// TIA Portal project "Palitizer" (V16)
// Vorlageprojekt für das Buch mit Zielsystem S7-1200

(* hardware
DEVICE "S7-1200-Station_1"  S7-1200 Station
   slot 0: "Baugruppenträger_0"  Rack  V1.0
   slot 1: "PLC_1"  CPU 1211C DC/DC/DC  6ES7 211-1AE40-0XB0  V4.1
DEVICE "HMI_1"  KTP700 Basic PN
   slot 0: "HMI_1"  KTP700 Basic PN  6AV2 123-2GB03-0AX0  16.0.0.0
   slot 1: "HMI_RT_1"  KTP700 Basic PN  6AV2 123-2GB03-0AX0  16.0.0.0
   slot 5: "HMI_1.IE_CP_1"  PROFINET Interface  16.0.0.0
      slot 1: "PROFINET Interface_1"  PROFINET Interface
         slot 1: "Port_1"  Port
*)

// ===== PLC "PLC_1"  CPU 1211C DC/DC/DC =====

VAR_GLOBAL   // PLC tag table "Standard-Variablentabelle"
   "I_Auto" AT %I0.0 : Bool;
   "I_Manual" AT %I0.1 : Bool;
   "I_Start" AT %I0.2 : Bool;
   "I_Stop" AT %I0.3 : Bool;
   "I_E_Stop" AT %I0.4 : Bool;
   "Q_Start_Light" AT %Q0.0 : Bool;
   "Q_Stop_Light" AT %Q0.1 : Bool;
   "M_Machine_Running" AT %M0.0 : Bool;
   "I_Pallet_Loaded" AT %I1.3 : Bool;   // Sensor ON the elevator. Goes TRUE when pallet is in position.
   "Q_Pallet_Feeder" AT %Q1.5 : Bool;   // The conveyor belt bringing pallets to the machine.
   "Q_Load_Pallet" AT %Q1.6 : Bool;   // The motorized rollers ON the elevator itself.
   "Q_Pallets_Emitter" AT %Q2.1 : Bool;   // Q_Pallets_Emitter
   "I_Box_At_Entry" AT %I0.6 : Bool;   // Photo-eye sensor that detects boxes passing.
   "I_Clamped" AT %I0.7 : Bool;   // Sensor confirming the clamp is fully closed.
   "Q_Box_Feeder" AT %Q0.4 : Bool;   // First conveyor bringing boxes in.
   "Q_Load_Belt" AT %Q0.5 : Bool;   // Second conveyor pushing boxes into the clamping area.
   "Q_Clamp" AT %Q0.7 : Bool;   // Pneumatic clamp to hold the row of boxes.
   "Q_Parts_Emitter" AT %Q2.0 : Bool;   // Spawns boxes in Factory I/O.
   "M_Box_Edge_Mem" AT %M0.1 : Bool;
   "M_Row_Ready" AT %M0.2 : Bool;
   "M_Reset_Row" AT %M0.3 : Bool;
   "Q_Push" AT %Q1.1 : Bool;   // Pushes clamped row onto plate
   "I_pusher_limit" AT %I1.0 : Bool;
   "Q_Open_Plate" AT %Q1.2 : Bool;
   "I_Plate_Limit" AT %I1.4 : Bool;
   "Q_Elevator_Up" AT %Q1.3 : Bool;
   "Q_Move_to_Limit" AT %Q1.4 : Bool;
   "I_Reset" AT %I1.5 : Bool;
   "Q_Elevator_down" AT %Q1.0 : Bool;
   "M_Eject_Pallet" AT %M0.4 : Bool;
   "I_Elevator_Moving" AT %I0.5 : Bool;
   "Q_Turn" AT %Q0.6 : Bool;
   "Q_Remover" AT %Q2.2 : Bool;
   "Q_Exit_Conveyor" AT %Q1.7 : Bool;
   "M_Target_Boxes" AT %MW10 : Int;   // Tells the counter how many boxes to wait for.
   "M_Target_Rows" AT %MW12 : Int;   // Tells the sequencer how many rows to push.
   "M_Enable_Turn" AT %M1.0 : Bool;   // Flag to activate the Turn actuator.
   "M_Machine_Fault" AT %M1.1 : Bool;
   "M_Cmd_Run" AT %M1.2 : Bool;
   "System_Byte" AT %MB5 : Byte;
   "FirstScan" AT %M5.0 : Bool;
   "DiagStatusUpdate" AT %M5.1 : Bool;
   "AlwaysTRUE" AT %M5.2 : Bool;
   "AlwaysFALSE" AT %M5.3 : Bool;
   "Clock_Byte" AT %MB2 : Byte;
   "Clock_10Hz" AT %M2.0 : Bool;
   "Clock_5Hz" AT %M2.1 : Bool;
   "Clock_2.5Hz" AT %M2.2 : Bool;
   "Clock_2Hz" AT %M2.3 : Bool;
   "Clock_1.25Hz" AT %M2.4 : Bool;
   "Clock_1Hz" AT %M2.5 : Bool;
   "Clock_0.625Hz" AT %M2.6 : Bool;
   "Clock_0.5Hz" AT %M2.7 : Bool;
   "Q_faulted" AT %Q0.2 : Bool;
   "Q_Warning_light" AT %Q2.3 : Bool;
   "negative_box_at_entry" AT %M0.5 : Bool;
   "Cmd_Push_Auto" AT %M0.6 : Bool;
   "Cmd_Push_Manual" AT %M0.7 : Bool;
   "Cmd_Clamp_Auto" AT %M3.0 : Bool;
   "Cmd_Clamp_Manual" AT %M3.1 : Bool;
   "Cmd_Plate_Auto" AT %M3.2 : Bool;
   "Cmd_Plate_Manual" AT %M3.3 : Bool;
   "Cmd_BoxFeed_Auto" AT %M3.4 : Bool;
   "Cmd_PalletFeed_Auto" AT %M3.5 : Bool;
   "Cmd_ExitConv_Auto" AT %M3.6 : Bool;
   "Cmd_BoxFeed_Manual" AT %M3.7 : Bool;
   "Cmd_PalletFeed_Manual" AT %M4.0 : Bool;
   "Cmd_ExitConv_Manual" AT %M4.1 : Bool;
   "Cmd_ElevUp_Auto" AT %M4.2 : Bool;
   "Cmd_ElevUp_Manual" AT %M4.3 : Bool;
   "Cmd_ElevDown_Auto" AT %M4.4 : Bool;
   "Cmd_ElevDown_Manual" AT %M4.5 : Bool;
   "System_Byte(1)" AT %MB1 : Byte;
   "Cmd_Turn_Auto" AT %M4.6 : Bool;
   "Cmd_Turn_Manual" AT %M4.7 : Bool;
   "I_Pallet_at_Entry" AT %I1.1 : Bool;
END_VAR

TYPE "UDT_SysCommand"
   STRUCT
      xSwAuto : Bool;
      xSwManual : Bool;
      xBtnStart : Bool;
      xBtnStop : Bool;
      xBtnReset : Bool;
      xEStop_OK : Bool;
      xHmiResetCounters : Bool;
      xHmiAckFault : Bool;
   END_STRUCT;
END_TYPE

TYPE "UDT_SysStatus"
   STRUCT
      xModeAuto : Bool;
      xModeManual : Bool;
      xRunning : Bool;
      xPaused : Bool;
      xFaulted : Bool;
      iStateID : Int;
      iCurrentLayer : Int;
      iTargetLayers : Int;
      iTotalBoxes : DInt;
      iTotalPallets : DInt;
      wAlarmWord : Word;
   END_STRUCT;
END_TYPE

DATA_BLOCK "FB1_Pallet_Handling_DB"   // DB1
{ S7_Optimized_Access := 'TRUE' }
VERSION : 0.1
// stored: InstanceOfName FB1_Pallet_Handling
"FB1_Pallet_Handling"
BEGIN
END_DATA_BLOCK

DATA_BLOCK "FB2_Box_Grouping_DB"   // DB3
{ S7_Optimized_Access := 'TRUE' }
VERSION : 0.1
// stored: InstanceOfName FB2_Box_Grouping
"FB2_Box_Grouping"
BEGIN
END_DATA_BLOCK

DATA_BLOCK "FB3_Elevator_Stacker_DB"   // DB5
{ S7_Optimized_Access := 'TRUE' }
VERSION : 0.1
// stored: InstanceOfName FB3_Elevator_Stacker
"FB3_Elevator_Stacker"
BEGIN
END_DATA_BLOCK

DATA_BLOCK "FB_ModeManager_DB"   // DB11
{ S7_Optimized_Access := 'TRUE' }
VERSION : 0.1
// stored: InstanceOfName FB_ModeManager
"FB_ModeManager"
BEGIN
END_DATA_BLOCK

DATA_BLOCK "DB_Machine"   // DB12
{ S7_Optimized_Access := 'FALSE' }
VERSION : 0.1
   VAR
      Cmd : "UDT_SysCommand";
      Sts : "UDT_SysStatus";
   END_VAR
BEGIN
END_DATA_BLOCK

DATA_BLOCK "InstDB_Cylinder_Pusher"   // DB13
{ S7_Optimized_Access := 'TRUE' }
VERSION : 0.1
// stored: InstanceOfName FB_Cylinder
"FB_Cylinder"
BEGIN
   i_xInterlock := true;
END_DATA_BLOCK

DATA_BLOCK "InstDB_Cyl_Clamp"   // DB14
{ S7_Optimized_Access := 'TRUE' }
VERSION : 0.1
// stored: InstanceOfName FB_Cylinder
"FB_Cylinder"
BEGIN
END_DATA_BLOCK

DATA_BLOCK "InstDB_Cyl_Plate"   // DB15
{ S7_Optimized_Access := 'TRUE' }
VERSION : 0.1
// stored: InstanceOfName FB_Cylinder
"FB_Cylinder"
BEGIN
END_DATA_BLOCK

DATA_BLOCK "FB_Motor_BoxFeed"   // DB16
{ S7_Optimized_Access := 'TRUE' }
VERSION : 0.1
// stored: InstanceOfName FB_Motor
"FB_Motor"
BEGIN
   i_xThermalFault := true;
END_DATA_BLOCK

DATA_BLOCK "FB_Motor_PalletFeed"   // DB17
{ S7_Optimized_Access := 'TRUE' }
VERSION : 0.1
// stored: InstanceOfName FB_Motor
"FB_Motor"
BEGIN
   i_xThermalFault := True;
END_DATA_BLOCK

DATA_BLOCK "FB_Motor_ExitConv"   // DB18
{ S7_Optimized_Access := 'TRUE' }
VERSION : 0.1
// stored: InstanceOfName FB_Motor
"FB_Motor"
BEGIN
   i_xThermalFault := true;
END_DATA_BLOCK

DATA_BLOCK "InstDB_Motor_ElevUp"   // DB19
{ S7_Optimized_Access := 'TRUE' }
VERSION : 0.1
// stored: InstanceOfName FB_Motor
"FB_Motor"
BEGIN
   i_xInterlock := true;
   i_xThermalFault := true;
END_DATA_BLOCK

DATA_BLOCK "InstDB_Motor_ElevDown"   // DB20
{ S7_Optimized_Access := 'TRUE' }
VERSION : 0.1
// stored: InstanceOfName FB_Motor
"FB_Motor"
BEGIN
   i_xThermalFault := true;
   i_xInterlock := true;
END_DATA_BLOCK

DATA_BLOCK "InstDB_Cyl_Turn"   // DB21
{ S7_Optimized_Access := 'TRUE' }
VERSION : 0.1
// stored: InstanceOfName FB_Cylinder
"FB_Cylinder"
BEGIN
END_DATA_BLOCK

// folder: System blocks/Program resources

DATA_BLOCK "counter1"   // DB2
{ S7_Optimized_Access := 'TRUE' }
AUTHOR : Simatic
FAMILY : IEC
NAME : CNTR
VERSION : 1.0
// stored: InstanceOfName IEC_COUNTER
"IEC_COUNTER"
BEGIN
END_DATA_BLOCK

DATA_BLOCK "IEC_Timer_0_DB"   // DB4
{ S7_Optimized_Access := 'TRUE' }
AUTHOR : Simatic
FAMILY : IEC
NAME : IEC_TMR
VERSION : 1.0
// stored: InstanceOfName IEC_TIMER
"IEC_TIMER"
BEGIN
END_DATA_BLOCK

DATA_BLOCK "IEC_Timer_0_DB_1"   // DB6
{ S7_Optimized_Access := 'TRUE' }
AUTHOR : Simatic
FAMILY : IEC
NAME : IEC_TMR
VERSION : 1.0
// stored: InstanceOfName IEC_TIMER
"IEC_TIMER"
BEGIN
END_DATA_BLOCK

DATA_BLOCK "IEC_Timer_0_DB_2"   // DB7
{ S7_Optimized_Access := 'TRUE' }
AUTHOR : Simatic
FAMILY : IEC
NAME : IEC_TMR
VERSION : 1.0
// stored: InstanceOfName IEC_TIMER
"IEC_TIMER"
BEGIN
END_DATA_BLOCK

DATA_BLOCK "plate_open"   // DB8
{ S7_Optimized_Access := 'TRUE' }
AUTHOR : Simatic
FAMILY : IEC
NAME : IEC_TMR
VERSION : 1.0
// stored: InstanceOfName IEC_TIMER
"IEC_TIMER"
BEGIN
END_DATA_BLOCK

DATA_BLOCK "plate_close"   // DB9
{ S7_Optimized_Access := 'TRUE' }
AUTHOR : Simatic
FAMILY : IEC
NAME : IEC_TMR
VERSION : 1.0
// stored: InstanceOfName IEC_TIMER
"IEC_TIMER"
BEGIN
END_DATA_BLOCK

DATA_BLOCK "Elevator_Timer"   // DB10
{ S7_Optimized_Access := 'TRUE' }
AUTHOR : Simatic
FAMILY : IEC
NAME : IEC_TMR
VERSION : 1.0
// stored: InstanceOfName IEC_TIMER
"IEC_TIMER"
BEGIN
END_DATA_BLOCK

// folder: (top level)

FUNCTION_BLOCK "FB1_Pallet_Handling"   // FB1, LAD
{ S7_Optimized_Access := 'TRUE' }
VERSION : 0.1
   VAR_INPUT
      i_stState : "UDT_SysStatus";
   END_VAR
BEGIN

REGION Network 1: Spawn Pallets
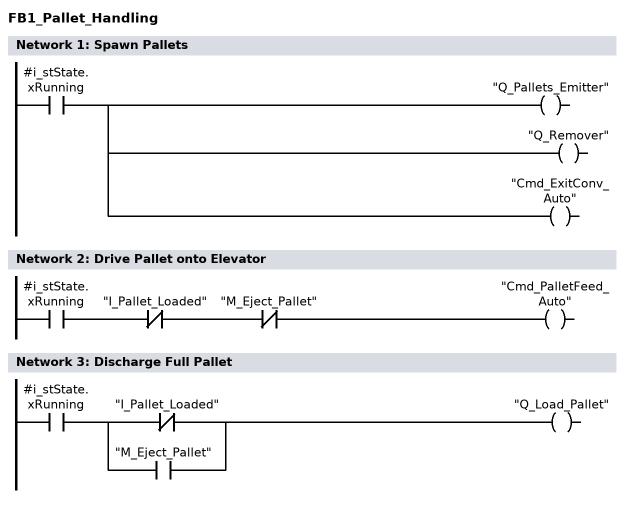
   RUNG wire#powerrail
      Contact( #i_stState.xRunning )
      wire#w1
      Coil( "Q_Pallets_Emitter" )
   END_RUNG
   RUNG wire#w1
      Coil( "Q_Remover" )
   END_RUNG
   RUNG wire#w1
      Coil( "Cmd_ExitConv_Auto" )
   END_RUNG
   // the same network as SCL:
   "Q_Pallets_Emitter" := #i_stState.xRunning;
   "Q_Remover" := #i_stState.xRunning;
   "Cmd_ExitConv_Auto" := #i_stState.xRunning;
END_REGION

REGION Network 2: Drive Pallet onto Elevator
   RUNG wire#powerrail
      Contact( #i_stState.xRunning )
      I_Contact( "I_Pallet_Loaded" )
      I_Contact( "M_Eject_Pallet" )
      Coil( "Cmd_PalletFeed_Auto" )
   END_RUNG
   // the same network as SCL:
   "Cmd_PalletFeed_Auto" := #i_stState.xRunning AND NOT "I_Pallet_Loaded" AND NOT "M_Eject_Pallet";
END_REGION

REGION Network 3: Discharge Full Pallet
   RUNG wire#powerrail
      Contact( #i_stState.xRunning )
      wire#w1
      I_Contact( "I_Pallet_Loaded" )
      wire#w2
      Coil( "Q_Load_Pallet" )
   END_RUNG
   RUNG wire#w1
      Contact( "M_Eject_Pallet" )
   END_RUNG wire#w2
   // the same network as SCL:
   "Q_Load_Pallet" := #i_stState.xRunning AND (NOT "I_Pallet_Loaded" OR "M_Eject_Pallet");
END_REGION
END_FUNCTION_BLOCK

FUNCTION_BLOCK "FB2_Box_Grouping"   // FB2, LAD
{ S7_Optimized_Access := 'TRUE' }
VERSION : 0.1
   VAR_INPUT
      i_stState : "UDT_SysStatus";
      i_stCmd : "UDT_SysCommand";
   END_VAR
   VAR_TEMP   // added for the SCL form of the ladder/FBD networks
      _w1 : Bool;
   END_VAR
BEGIN

REGION Network 1: Spawns boxes in Factory I/O.
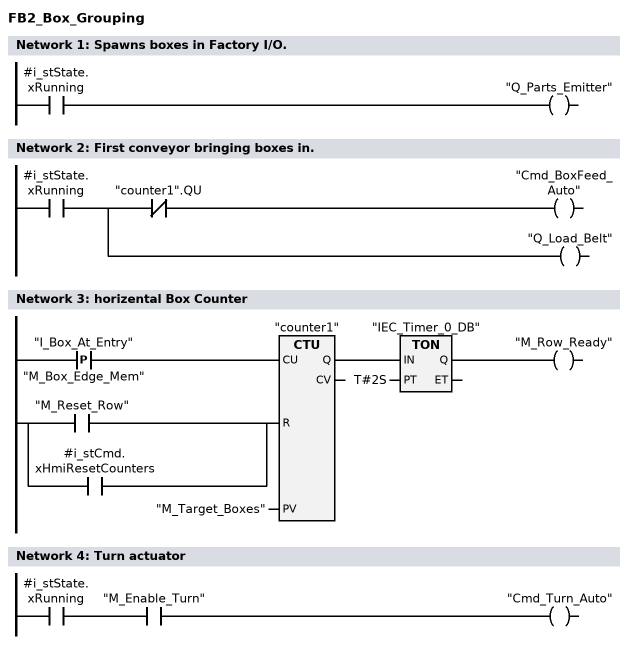
   RUNG wire#powerrail
      Contact( #i_stState.xRunning )
      Coil( "Q_Parts_Emitter" )
   END_RUNG
   // the same network as SCL:
   "Q_Parts_Emitter" := #i_stState.xRunning;
END_REGION

REGION Network 2: First conveyor bringing boxes in.
   RUNG wire#powerrail
      Contact( #i_stState.xRunning )
      wire#w1
      I_Contact( "counter1".QU )
      Coil( "Cmd_BoxFeed_Auto" )
   END_RUNG
   RUNG wire#w1
      Coil( "Q_Load_Belt" )
   END_RUNG
   // the same network as SCL:
   "Cmd_BoxFeed_Auto" := #i_stState.xRunning AND NOT "counter1".QU;
   "Q_Load_Belt" := #i_stState.xRunning;
END_REGION

REGION Network 3: horizental Box Counter
   #_w1 := "I_Box_At_Entry" AND NOT "M_Box_Edge_Mem";   // rising edge of "I_Box_At_Entry"
   "M_Box_Edge_Mem" := "I_Box_At_Entry";
   "counter1".CTU(CU := #_w1, R := "M_Reset_Row" OR #i_stCmd.xHmiResetCounters, PV := "M_Target_Boxes");
   "IEC_Timer_0_DB".TON(IN := "counter1".Q, PT := T#2S);
   "M_Row_Ready" := "IEC_Timer_0_DB".Q;
END_REGION

REGION Network 4: Turn actuator
   RUNG wire#powerrail
      Contact( #i_stState.xRunning )
      Contact( "M_Enable_Turn" )
      Coil( "Cmd_Turn_Auto" )
   END_RUNG
   // the same network as SCL:
   "Cmd_Turn_Auto" := #i_stState.xRunning AND "M_Enable_Turn";
END_REGION
END_FUNCTION_BLOCK

FUNCTION_BLOCK "FB3_Elevator_Stacker"   // FB3, SCL
{ S7_Optimized_Access := 'TRUE' }
VERSION : 0.1
   VAR_INPUT
      i_stState : "UDT_SysStatus";
      i_stCmd : "UDT_SysCommand";
   END_VAR
   VAR_IN_OUT
      io_stState : "UDT_SysStatus";
   END_VAR
   VAR
      stat_Step : Int;
      stat_Retract_Timer : IEC_TIMER;
      stat_Row_Count : Int;
      stat_horizental_box_count : Int;
      stat_vertical_box_count : Int;
      stat_Box_Count : Int;
      stat_Layer_Count : Int;
      stat_Target_Boxes : Int;
      stat_Target_Rows : Int;
      stat_Box_Sensor_Prev : Bool;
      stat_Fault_ID : Int;
      stat_Push_Timeout : IEC_TIMER;
      stat_Plate_Timeout : IEC_TIMER;
      stat_Eject_Timeout : IEC_TIMER;
      push : TON_TIME;
      EjectTimeout : TON_TIME;
   END_VAR
BEGIN
   // --- 1. Fault Reset Logic ---
   // Operator must clear the jam and press Reset to clear the Fault ID
   IF ("I_Reset" OR #i_stCmd.xHmiAckFault)  AND "I_E_Stop" THEN
       #stat_Fault_ID := 0;
       "M_Machine_Fault" := FALSE;
   END_IF;
   // --- 2. Diagnostics & Watchdog Timers ---
   // E-Stop Monitor
   IF NOT "I_E_Stop" THEN
       #stat_Fault_ID := 1;
       #io_stState.xFaulted := TRUE;
       #stat_Step := 0;
   END_IF;
   // Watchdog Timers (Running parallel to the state machine)
   #push(IN:=#stat_Step = 10,
         PT:=T#2.0S);

   #EjectTimeout(IN := #stat_Step = 81,
                 PT := T#8.0S);


   #stat_Plate_Timeout.IN := #stat_Step = 60;
   #stat_Plate_Timeout.PT := T#4.0S;

   // Fault Triggers (If a timer finishes, assign the specific Fault ID)
   IF #push.Q THEN
       #stat_Fault_ID := 2;
       #io_stState.xFaulted := TRUE;
       #stat_Step := 0;
   END_IF;
   IF #stat_Plate_Timeout.Q THEN
       #stat_Fault_ID := 3;
       #io_stState.xFaulted := TRUE;
       #stat_Step := 0;
   END_IF;
   IF #EjectTimeout.Q THEN
       #stat_Fault_ID := 4;
       #io_stState.xFaulted := TRUE;
       #stat_Step := 0;
   END_IF;
   // --- Alarm Word Mapping (Slice Access) ---
   // If the Fault ID equals 1, turn on Bit 1 of the Word.
   #io_stState.wAlarmWord.%X1 := (#stat_Fault_ID = 1);
   #io_stState.wAlarmWord.%X2 := (#stat_Fault_ID = 2);
   #io_stState.wAlarmWord.%X3 := (#stat_Fault_ID = 3);
   #io_stState.wAlarmWord.%X4 := (#stat_Fault_ID = 4);
   // --- Safety & Mode Interlock ---
   IF NOT #i_stState.xRunning THEN

       "Cmd_Push_Auto" := FALSE;
       "Cmd_Plate_Auto" := FALSE;
       "Cmd_ElevUp_Auto" := FALSE;
       "Cmd_ElevDown_Auto" := FALSE;
       "Q_Move_to_Limit" := FALSE;
       "M_Reset_Row" := FALSE;
       "M_Eject_Pallet" := FALSE;
       "Cmd_Clamp_Auto" := FALSE;
       #stat_Row_Count := 0;
       #stat_Layer_Count := 0;
       RETURN;
   END_IF;
   // --- Maintenance Reset ---
   IF #i_stCmd.xHmiResetCounters THEN
       #stat_Layer_Count := 0;
       #stat_Row_Count := 0;
       #io_stState.iTotalBoxes := 0;
       #io_stState.iTotalPallets := 0;
       #stat_Step := 0; // Safely drops the machine back to the IDLE state
   END_IF;

   // --- Timer Execution ---
   "IEC_Timer_0_DB_1".TON(IN := (#stat_Step = 20),
                          PT := T#1.5S); // Retract
   "IEC_Timer_0_DB_2".TON(IN := (#stat_Step = 10),
                          PT := T#0.5S); // Push
   "plate_open".TON(IN := (#stat_Step = 40),
                    PT := T#3.0S); // Plate open
   "plate_close".TON(IN := (#stat_Step = 60),
                     PT := T#2.0S); // plate close
   "Elevator_Timer".TON(IN := (#stat_Step = 52),
                        PT := T#500MS);
   // --- Dynamic Pattern Generator ---
   // Even Layers (0, 2): 3 boxes per row, 2 rows. TURN OFF.
   IF (#stat_Layer_Count MOD 2) = 0 THEN
       "M_Target_Boxes" := 2;
       "M_Target_Rows" := 3;
       "M_Enable_Turn" := FALSE;
       // Odd Layers (1, 3): 2 boxes per row, 3 rows. TURN ON.
   ELSE
       "M_Target_Boxes" := 3;
       "M_Target_Rows" := 2;
       "M_Enable_Turn" := TRUE;
   END_IF;

   // --- The Core State Machine ---
   CASE #stat_Step OF

       0:  // IDLE STATE
           "Cmd_Push_Auto" := FALSE;
           "M_Reset_Row" := FALSE;
           "Cmd_Plate_Auto" := FALSE;
           "Cmd_ElevUp_Auto" := FALSE;
           "Cmd_ElevDown_Auto" := FALSE;
           "Q_Move_to_Limit" := FALSE;
           "M_Eject_Pallet" := FALSE;

           // Force the elevator to absolute top for a fresh pallet
           IF #stat_Layer_Count = 0 AND "I_Pallet_Loaded" THEN
               "Q_Move_to_Limit" := TRUE;
               "Cmd_ElevUp_Auto" := TRUE;
           END_IF;

           // Proceed ONLY if row is ready, pallet is present, and elevator is at the top
           IF "M_Row_Ready" AND "I_Pallet_Loaded" AND NOT "I_Elevator_Moving" THEN
               "Q_Move_to_Limit" := FALSE;
               "Cmd_ElevUp_Auto" := FALSE;
               // FIXED: Removed premature Elevator Down command here
               #stat_Step := 10;
           END_IF;

       10: // PUSH STATE
           "Q_Box_Feeder" := FALSE;
           "Cmd_Push_Auto" := TRUE;

           IF "IEC_Timer_0_DB_2".Q THEN
               #stat_Step := 20;
           END_IF;

       20: // RETRACT STATE
           "Q_Box_Feeder" := FALSE;
           "Cmd_Push_Auto" := FALSE;
           "M_Reset_Row" := TRUE;

           IF "IEC_Timer_0_DB_1".Q THEN
               #stat_Step := 30;
           END_IF;

       30: // ROW MATH (FIXED: Single Scan Execution)
           "Q_Box_Feeder" := TRUE;
           "M_Reset_Row" := FALSE;
           #stat_Row_Count := #stat_Row_Count + 1; // Increment happens exactly once
           // Add boxes to the total 
           #io_stState.iTotalBoxes := #io_stState.iTotalBoxes + "M_Target_Boxes";
           IF #stat_Row_Count >= "M_Target_Rows" THEN
               #stat_Layer_Count := #stat_Layer_Count + 1;
               #stat_Step := 31; // Jump to new state to wait for clamp
           ELSE
               #stat_Step := 0;  // Go back for next row
           END_IF;

       31: // WAIT FOR CLAMP (Prevents Math Loop Bug)
           "Cmd_Clamp_Auto" := TRUE;

           IF "I_Clamped" THEN
               #stat_Step := 40;
           END_IF;

       40: // DROP LAYER (OPEN PLATE)
           "Cmd_Clamp_Auto" := TRUE;

           "Cmd_Plate_Auto" := TRUE;

           IF "plate_open".Q THEN

               #stat_Step := 50;
           END_IF;

       50: // INDEX 1 START (FIXED: Race condition protection restored)
           "Cmd_ElevUp_Auto" := FALSE;
           "Q_Move_to_Limit" := FALSE;
           "Cmd_ElevDown_Auto" := TRUE;

           IF "I_Elevator_Moving" THEN // Wait for motor to physically start
               #stat_Step := 51;
           END_IF;

       51: // INDEX 1 FINISH 
           IF NOT "I_Elevator_Moving" THEN
               "Cmd_ElevDown_Auto" := FALSE;
               #stat_Step := 52;
           END_IF;

       52: // PAUSE 
           IF "Elevator_Timer".Q THEN
               #stat_Step := 54;
           END_IF;

       53: // INDEX 2 START 
           "Cmd_ElevDown_Auto" := TRUE;
           IF "I_Elevator_Moving" THEN
               #stat_Step := 54;
           END_IF;

       54: // INDEX 2 FINISH
           IF NOT "I_Elevator_Moving" THEN
               "Cmd_ElevDown_Auto" := FALSE;
               #stat_Step := 60;
           END_IF;

       60: // CLOSE PLATE 
           "Cmd_Plate_Auto" := FALSE;
           IF "plate_close".Q THEN
               "Cmd_Clamp_Auto" := FALSE;
               #stat_Row_Count := 0;
               // "M_Reset_Row" := TRUE;
               #stat_Step := 70;
           END_IF;

       70: // LAYER DECISION 
           IF #stat_Layer_Count >= 4 THEN
               #stat_Step := 80;
           ELSE
               #stat_Step := 0;
           END_IF;

       80: // DISCHARGE PALLET (FIXED: Race condition protection restored)
           "Q_Move_to_Limit" := TRUE;
           "Cmd_ElevDown_Auto" := TRUE;

           IF "I_Elevator_Moving" THEN // Wait for motor to start
               #stat_Step := 81;
           END_IF;

       81: // WAIT FOR DISCHARGE 
           IF NOT "I_Elevator_Moving" THEN
               "M_Eject_Pallet" := TRUE;
               "Cmd_ElevDown_Auto" := FALSE;
               "Q_Move_to_Limit" := FALSE;

               IF NOT "I_Pallet_Loaded" THEN
                   #stat_Layer_Count := 0;
                   "M_Eject_Pallet" := FALSE;
                   #stat_Step := 0;
                   #io_stState.iTotalPallets := #io_stState.iTotalPallets + 1;
               END_IF;
           END_IF;

   END_CASE;

   // --- HMI Data Reporting ---
   #io_stState.iCurrentLayer := #stat_Layer_Count;
   #io_stState.iTargetLayers := 4; // Since  logic ejects at layer 4
END_FUNCTION_BLOCK

FUNCTION_BLOCK "FB_ModeManager"   // FB4, SCL
{ S7_Optimized_Access := 'TRUE' }
VERSION : 0.1
   VAR_IN_OUT
      io_Cmd : "UDT_SysCommand";
      io_Sts : "UDT_SysStatus";
   END_VAR
BEGIN
   // --- 1. Master Safety Override ---
   // If the E-stop is pressed, immediately kill the run and trigger a fault.
   IF NOT #io_Cmd.xEStop_OK THEN
       #io_Sts.xFaulted := TRUE;
       #io_Sts.xRunning := FALSE;
   END_IF;

   // Fault reset logic 
   IF #io_Cmd.xBtnReset AND #io_Cmd.xEStop_OK THEN
       #io_Sts.xFaulted := FALSE;
   END_IF;

   // --- 2.Mode selection --- 
   // Determine machine mode based on physical switch 
   IF #io_Cmd.xSwAuto AND NOT #io_Sts.xFaulted THEN
       #io_Sts.xModeAuto := TRUE;
       #io_Sts.xModeManual := FALSE;

   ELSIF #io_Cmd.xSwManual AND NOT #io_Sts.xFaulted THEN
       #io_Sts.xModeAuto := FALSE;
       #io_Sts.xModeManual := TRUE;
       #io_Sts.xRunning := FALSE; // Instantly drop the run permissive if dropping out of Auto

   ELSE
       #io_Sts.xModeAuto := FALSE;
       #io_Sts.xModeManual := FALSE;
       #io_Sts.xRunning := FALSE;
   END_IF;

   // --- 3. Start / Stop Latch (Auto Mode Only) ---
   IF #io_Sts.xModeAuto THEN
       // start sequence 
       IF #io_Cmd.xBtnStart THEN
           #io_Sts.xRunning := TRUE;
       END_IF;

       // Hold sequence pause 
       IF NOT #io_Cmd.xBtnStop THEN
           #io_Sts.xRunning := FALSE;
       END_IF;

   END_IF;

   // --- 4. HMI State & Indicator Logic ---
   IF #io_Sts.xFaulted THEN
       #io_Sts.iStateID := 5; // Faulted 
   ELSIF #io_Sts.xModeManual THEN
       #io_Sts.iStateID := 4; // manual mode 
   ELSIF #io_Sts.xModeAuto AND #io_Sts.xRunning THEN
       #io_Sts.iStateID := 2; // auto mode running 
   ELSIF #io_Sts.xModeAuto AND NOT #io_Sts.xRunning THEN
       #io_Sts.iStateID := 3; // auto mode paused 
   ELSE
       #io_Sts.iStateID := 1; // idle 
   END_IF;

   // Indicator Light Flag (TRUE when paused in Auto or waiting in Manual)
   #io_Sts.xPaused := (#io_Sts.iStateID = 3) OR (#io_Sts.iStateID = 4);
END_FUNCTION_BLOCK

FUNCTION_BLOCK "FB_Cylinder"   // FB5, SCL
{ S7_Optimized_Access := 'TRUE' }
VERSION : 0.1
   VAR_INPUT
      i_stState : "UDT_SysStatus";   // The master mode from DB_Machine.
      i_xAutoCmd : Bool;   // The command from FB3 sequencer
      i_xManualCmd : Bool;   // he jog button from the operator.
      i_xInterlock : Bool := True;   // Safety condition
   END_VAR
   VAR_OUTPUT
      q_xValveOut : Bool;   // The signal going to the physical coil
   END_VAR
BEGIN
   // Check safety interlock first
   IF #i_xInterlock THEN
       // Auto mode : listen to the sequencer 
       IF #i_stState.xModeAuto AND #i_stState.xRunning THEN
           #q_xValveOut := #i_xAutoCmd;
           // MANUAL MODE: Listen strictly to the operator
       ELSIF #i_stState.xModeManual THEN
           #q_xValveOut := #i_xManualCmd;
           // OFF / FAULTED: Drop output for safet
       ELSE
           #q_xValveOut := FALSE;
       END_IF;
   ELSE
       #q_xValveOut := FALSE;
   END_IF;
END_FUNCTION_BLOCK

FUNCTION_BLOCK "FB_Motor"   // FB6, SCL
{ S7_Optimized_Access := 'TRUE' }
VERSION : 0.1
   VAR_INPUT
      i_stState : "UDT_SysStatus";
      i_xAutoCmd : Bool;
      i_xManualCmd : Bool;
      i_xInterlock : Bool;
      i_xThermalFault : Bool;
   END_VAR
   VAR_OUTPUT
      q_xRunFwd : Bool;
   END_VAR
BEGIN
   // Check motor hardware health first (assuming NC thermal contact)
   IF #i_xThermalFault THEN

       // check mechanical interlock 
       IF #i_xInterlock THEN

           // auto mode 
           IF #i_stState.xModeAuto AND #i_stState.xRunning THEN
               #q_xRunFwd := #i_xAutoCmd;

               // manual mode 
           ELSIF #i_stState.xModeManual THEN
               #q_xRunFwd := #i_xManualCmd;

               // off / faulted 
           ELSE
               #q_xRunFwd := FALSE;
           END_IF;
       ELSE
           // Interlock broken
           #q_xRunFwd := FALSE;
       END_IF;
   ELSE
       // Motor thermal overload tripped!
       #q_xRunFwd := FALSE;
   END_IF;
END_FUNCTION_BLOCK

FUNCTION "MHJ-PLC-Lab-Function-S71200" : Void   // FC9000, SCL
{ S7_Optimized_Access := 'TRUE' }
VERSION : 0.1
   VAR_TEMP
      rdTimeReturn : Int;
      outputTime : DTL;
      SyncVal : Byte;
      forVal : Int;
      forVal_2 : Int;
      Value : Byte;
   END_VAR
   VAR CONSTANT
      CompVal : Byte := 16#34;
      Value_01 : Byte := 16#11;
      Value_01_DW : DWord := 16#A165_D992;
      Value_02_DW : DWord := 16#58BE_4401;
   END_VAR
BEGIN

   #Value:=PEEK(area := 16#82,
        dbNumber := 0,
        byteOffset := 511);
   #Value := #Value + 1;

   POKE(area := 16#82,
        dbNumber := 0,
        byteOffset := 511,
        value := #Value);

   POKE(area:=16#81,
        dbNumber:=0,
        byteOffset:=1016,
        value:=#Value_01_DW);
   POKE(area := 16#81,
        dbNumber := 0,
        byteOffset := 1020,
        value := #Value_02_DW);

   POKE(area := 16#81,
        dbNumber := 0,
        byteOffset := 511,
        value := B#16#00);

   FOR #forVal := 0 TO 120 DO
       FOR #forVal_2:=0 TO 10 DO
           #rdTimeReturn:=RD_SYS_T(#outputTime);
           #rdTimeReturn := WR_SYS_T(#outputTime);
           #rdTimeReturn := RD_SYS_T(#outputTime);
           #rdTimeReturn := WR_SYS_T(#outputTime);
       END_FOR;
       #SyncVal:= PEEK(area := 16#81,
                      dbNumber := 0,
                      byteOffset := 511);
       IF #SyncVal = #CompVal THEN
          GOTO M_1;
       END_IF;
   END_FOR;
   RETURN;

   M_1:
   POKE(area := 16#81,
        dbNumber := 0,
        byteOffset := 511,
        value := B#16#0);
END_FUNCTION

ORGANIZATION_BLOCK "Main"   // OB1, LAD, ProgramCycle
TITLE = "Main Program Sweep (Cycle)"
{ S7_Optimized_Access := 'TRUE' }
VERSION : 0.1
   VAR_INPUT
      Initial_Call : Bool;   // Initial call of this OB
      Remanence : Bool;   // =True, if remanent data are available
   END_VAR
   VAR_TEMP
      Start : Bool;
      ne_palet_at_entry : Bool;
      palet_loaded_pe : Bool;
   END_VAR
BEGIN

REGION Network 1: Konnektierungsbaustein für PLC-Lab
   // Im Netzwerk 1 wird der Konnektierungsbaustein für PLC-Lab aufgerufen.
   // Dieser Aufruf darf nicht entfernt werden!
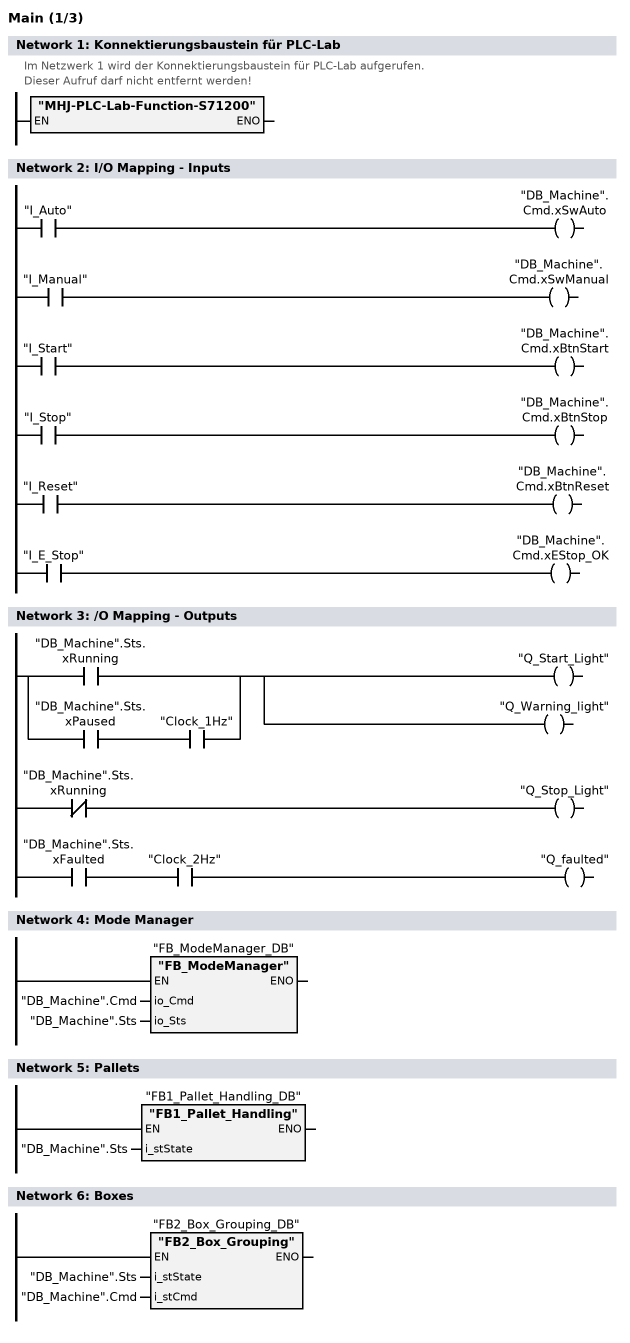
   RUNG wire#powerrail
      "MHJ-PLC-Lab-Function-S71200"()
   END_RUNG
   // the same network as SCL:
   "MHJ-PLC-Lab-Function-S71200"();
END_REGION

REGION Network 2: I/O Mapping - Inputs
   RUNG wire#powerrail
      Contact( "I_Auto" )
      Coil( "DB_Machine".Cmd.xSwAuto )
   END_RUNG
   RUNG wire#powerrail
      Contact( "I_Manual" )
      Coil( "DB_Machine".Cmd.xSwManual )
   END_RUNG
   RUNG wire#powerrail
      Contact( "I_Start" )
      Coil( "DB_Machine".Cmd.xBtnStart )
   END_RUNG
   RUNG wire#powerrail
      Contact( "I_Stop" )
      Coil( "DB_Machine".Cmd.xBtnStop )
   END_RUNG
   RUNG wire#powerrail
      Contact( "I_Reset" )
      Coil( "DB_Machine".Cmd.xBtnReset )
   END_RUNG
   RUNG wire#powerrail
      Contact( "I_E_Stop" )
      Coil( "DB_Machine".Cmd.xEStop_OK )
   END_RUNG
   // the same network as SCL:
   "DB_Machine".Cmd.xSwAuto := "I_Auto";
   "DB_Machine".Cmd.xSwManual := "I_Manual";
   "DB_Machine".Cmd.xBtnStart := "I_Start";
   "DB_Machine".Cmd.xBtnStop := "I_Stop";
   "DB_Machine".Cmd.xBtnReset := "I_Reset";
   "DB_Machine".Cmd.xEStop_OK := "I_E_Stop";
END_REGION

REGION Network 3: /O Mapping - Outputs
   RUNG wire#powerrail
      Contact( "DB_Machine".Sts.xRunning )
      wire#w1
      Coil( "Q_Start_Light" )
   END_RUNG
   RUNG wire#powerrail
      Contact( "DB_Machine".Sts.xPaused )
      Contact( "Clock_1Hz" )
   END_RUNG wire#w1
   RUNG wire#w1
      Coil( "Q_Warning_light" )
   END_RUNG
   RUNG wire#powerrail
      I_Contact( "DB_Machine".Sts.xRunning )
      Coil( "Q_Stop_Light" )
   END_RUNG
   RUNG wire#powerrail
      Contact( "DB_Machine".Sts.xFaulted )
      Contact( "Clock_2Hz" )
      Coil( "Q_faulted" )
   END_RUNG
   // the same network as SCL:
   "Q_Start_Light" := "DB_Machine".Sts.xRunning OR ("DB_Machine".Sts.xPaused AND "Clock_1Hz");
   "Q_Warning_light" := "Q_Start_Light";
   "Q_Stop_Light" := NOT "DB_Machine".Sts.xRunning;
   "Q_faulted" := "DB_Machine".Sts.xFaulted AND "Clock_2Hz";
END_REGION

REGION Network 4: Mode Manager
   RUNG wire#powerrail
      "FB_ModeManager_DB"(io_Cmd := "DB_Machine".Cmd, io_Sts := "DB_Machine".Sts)
   END_RUNG
   // the same network as SCL:
   "FB_ModeManager_DB"(io_Cmd := "DB_Machine".Cmd, io_Sts := "DB_Machine".Sts);   // "FB_ModeManager"
END_REGION

REGION Network 5: Pallets
   RUNG wire#powerrail
      "FB1_Pallet_Handling_DB"(i_stState := "DB_Machine".Sts)
   END_RUNG
   // the same network as SCL:
   "FB1_Pallet_Handling_DB"(i_stState := "DB_Machine".Sts);   // "FB1_Pallet_Handling"
END_REGION

REGION Network 6: Boxes
   RUNG wire#powerrail
      "FB2_Box_Grouping_DB"(i_stState := "DB_Machine".Sts, i_stCmd := "DB_Machine".Cmd)
   END_RUNG
   // the same network as SCL:
   "FB2_Box_Grouping_DB"(i_stState := "DB_Machine".Sts, i_stCmd := "DB_Machine".Cmd);   // "FB2_Box_Grouping"
END_REGION

REGION Network 7
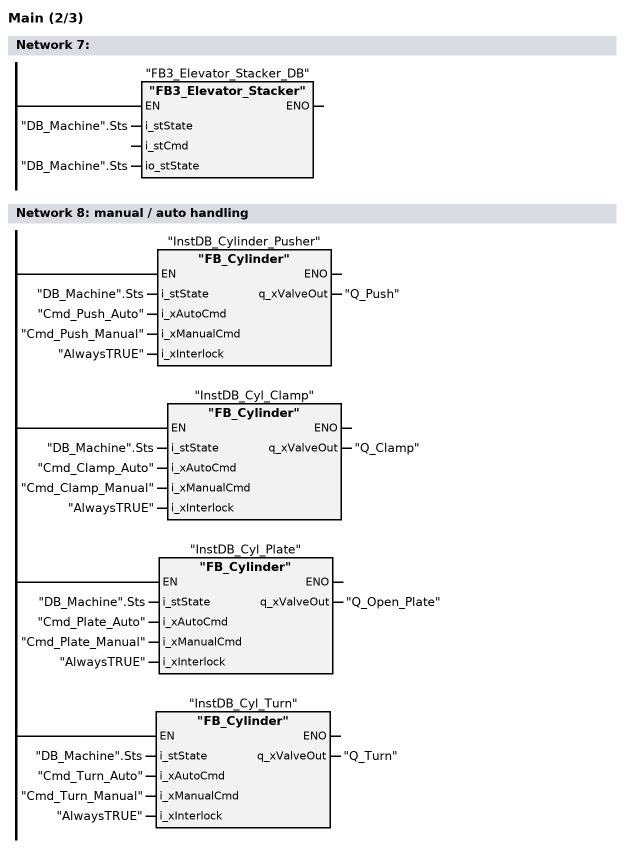
   RUNG wire#powerrail
      "FB3_Elevator_Stacker_DB"(i_stState := "DB_Machine".Sts, i_stCmd :=, io_stState := "DB_Machine".Sts)
   END_RUNG
   // the same network as SCL:
   "FB3_Elevator_Stacker_DB"(i_stState := "DB_Machine".Sts, io_stState := "DB_Machine".Sts);   // "FB3_Elevator_Stacker"
END_REGION

REGION Network 8: manual / auto handling
   RUNG wire#powerrail
      "InstDB_Cylinder_Pusher"(i_stState := "DB_Machine".Sts, i_xAutoCmd := "Cmd_Push_Auto", i_xManualCmd := "Cmd_Push_Manual", i_xInterlock := "AlwaysTRUE", q_xValveOut => "Q_Push")
   END_RUNG
   RUNG wire#powerrail
      "InstDB_Cyl_Clamp"(i_stState := "DB_Machine".Sts, i_xAutoCmd := "Cmd_Clamp_Auto", i_xManualCmd := "Cmd_Clamp_Manual", i_xInterlock := "AlwaysTRUE", q_xValveOut => "Q_Clamp")
   END_RUNG
   RUNG wire#powerrail
      "InstDB_Cyl_Plate"(i_stState := "DB_Machine".Sts, i_xAutoCmd := "Cmd_Plate_Auto", i_xManualCmd := "Cmd_Plate_Manual", i_xInterlock := "AlwaysTRUE", q_xValveOut => "Q_Open_Plate")
   END_RUNG
   RUNG wire#powerrail
      "InstDB_Cyl_Turn"(i_stState := "DB_Machine".Sts, i_xAutoCmd := "Cmd_Turn_Auto", i_xManualCmd := "Cmd_Turn_Manual", i_xInterlock := "AlwaysTRUE", q_xValveOut => "Q_Turn")
   END_RUNG
   // the same network as SCL:
   "InstDB_Cylinder_Pusher"(i_stState := "DB_Machine".Sts,   // "FB_Cylinder"
                           i_xAutoCmd := "Cmd_Push_Auto",
                           i_xManualCmd := "Cmd_Push_Manual",
                           i_xInterlock := "AlwaysTRUE",
                           q_xValveOut => "Q_Push");
   "InstDB_Cyl_Clamp"(i_stState := "DB_Machine".Sts,   // "FB_Cylinder"
                      i_xAutoCmd := "Cmd_Clamp_Auto",
                      i_xManualCmd := "Cmd_Clamp_Manual",
                      i_xInterlock := "AlwaysTRUE",
                      q_xValveOut => "Q_Clamp");
   "InstDB_Cyl_Plate"(i_stState := "DB_Machine".Sts,   // "FB_Cylinder"
                      i_xAutoCmd := "Cmd_Plate_Auto",
                      i_xManualCmd := "Cmd_Plate_Manual",
                      i_xInterlock := "AlwaysTRUE",
                      q_xValveOut => "Q_Open_Plate");
   "InstDB_Cyl_Turn"(i_stState := "DB_Machine".Sts,   // "FB_Cylinder"
                     i_xAutoCmd := "Cmd_Turn_Auto",
                     i_xManualCmd := "Cmd_Turn_Manual",
                     i_xInterlock := "AlwaysTRUE",
                     q_xValveOut => "Q_Turn");
END_REGION

REGION Network 9: motors manual/auto
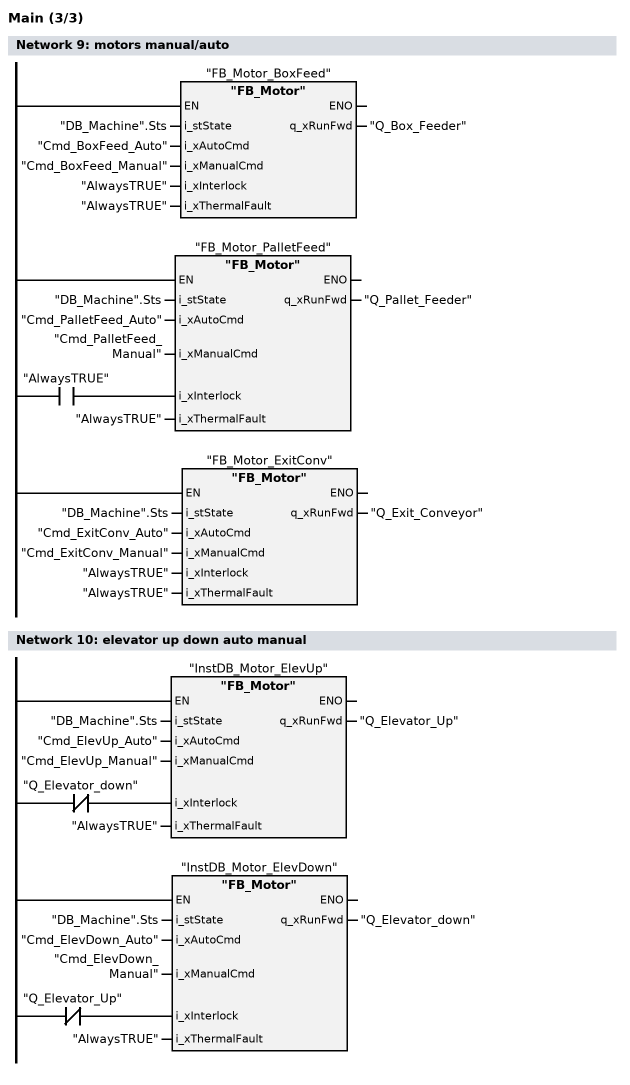
   RUNG wire#powerrail
      "FB_Motor_BoxFeed"(i_stState := "DB_Machine".Sts, i_xAutoCmd := "Cmd_BoxFeed_Auto", i_xManualCmd := "Cmd_BoxFeed_Manual", i_xInterlock := "AlwaysTRUE", i_xThermalFault := "AlwaysTRUE", q_xRunFwd => "Q_Box_Feeder")
   END_RUNG
   RUNG wire#powerrail
      "FB_Motor_PalletFeed"(i_xInterlock := wire#w1, i_stState := "DB_Machine".Sts, i_xAutoCmd := "Cmd_PalletFeed_Auto", i_xManualCmd := "Cmd_PalletFeed_Manual", i_xThermalFault := "AlwaysTRUE", q_xRunFwd => "Q_Pallet_Feeder")
   END_RUNG
   RUNG wire#powerrail
      Contact( "AlwaysTRUE" )
   END_RUNG wire#w1
   RUNG wire#powerrail
      "FB_Motor_ExitConv"(i_stState := "DB_Machine".Sts, i_xAutoCmd := "Cmd_ExitConv_Auto", i_xManualCmd := "Cmd_ExitConv_Manual", i_xInterlock := "AlwaysTRUE", i_xThermalFault := "AlwaysTRUE", q_xRunFwd => "Q_Exit_Conveyor")
   END_RUNG
   // the same network as SCL:
   "FB_Motor_BoxFeed"(i_stState := "DB_Machine".Sts,   // "FB_Motor"
                      i_xAutoCmd := "Cmd_BoxFeed_Auto",
                      i_xManualCmd := "Cmd_BoxFeed_Manual",
                      i_xInterlock := "AlwaysTRUE",
                      i_xThermalFault := "AlwaysTRUE",
                      q_xRunFwd => "Q_Box_Feeder");
   "FB_Motor_PalletFeed"(i_stState := "DB_Machine".Sts,   // "FB_Motor"
                         i_xAutoCmd := "Cmd_PalletFeed_Auto",
                         i_xManualCmd := "Cmd_PalletFeed_Manual",
                         i_xInterlock := "AlwaysTRUE",
                         i_xThermalFault := "AlwaysTRUE",
                         q_xRunFwd => "Q_Pallet_Feeder");
   "FB_Motor_ExitConv"(i_stState := "DB_Machine".Sts,   // "FB_Motor"
                       i_xAutoCmd := "Cmd_ExitConv_Auto",
                       i_xManualCmd := "Cmd_ExitConv_Manual",
                       i_xInterlock := "AlwaysTRUE",
                       i_xThermalFault := "AlwaysTRUE",
                       q_xRunFwd => "Q_Exit_Conveyor");
END_REGION

REGION Network 10: elevator up down auto manual
   RUNG wire#powerrail
      "InstDB_Motor_ElevUp"(i_xInterlock := wire#w1, i_stState := "DB_Machine".Sts, i_xAutoCmd := "Cmd_ElevUp_Auto", i_xManualCmd := "Cmd_ElevUp_Manual", i_xThermalFault := "AlwaysTRUE", q_xRunFwd => "Q_Elevator_Up")
   END_RUNG
   RUNG wire#powerrail
      I_Contact( "Q_Elevator_down" )
   END_RUNG wire#w1
   RUNG wire#powerrail
      "InstDB_Motor_ElevDown"(i_xInterlock := wire#w2, i_stState := "DB_Machine".Sts, i_xAutoCmd := "Cmd_ElevDown_Auto", i_xManualCmd := "Cmd_ElevDown_Manual", i_xThermalFault := "AlwaysTRUE", q_xRunFwd => "Q_Elevator_down")
   END_RUNG
   RUNG wire#powerrail
      I_Contact( "Q_Elevator_Up" )
   END_RUNG wire#w2
   // the same network as SCL:
   "InstDB_Motor_ElevUp"(i_stState := "DB_Machine".Sts,   // "FB_Motor"
                         i_xAutoCmd := "Cmd_ElevUp_Auto",
                         i_xManualCmd := "Cmd_ElevUp_Manual",
                         i_xInterlock := NOT "Q_Elevator_down",
                         i_xThermalFault := "AlwaysTRUE",
                         q_xRunFwd => "Q_Elevator_Up");
   "InstDB_Motor_ElevDown"(i_stState := "DB_Machine".Sts,   // "FB_Motor"
                           i_xAutoCmd := "Cmd_ElevDown_Auto",
                           i_xManualCmd := "Cmd_ElevDown_Manual",
                           i_xInterlock := NOT "Q_Elevator_Up",
                           i_xThermalFault := "AlwaysTRUE",
                           q_xRunFwd => "Q_Elevator_down");
END_REGION
END_ORGANIZATION_BLOCK

(* ===== HMI "HMI_RT_1" =====
system functions are stored by id; their names below are inferred from use
connection "HMI_Connection_1": ETHERNET, SMART_S7_1200_OMS

HMI tags "Default tag table"
   "Tag_ScreenNumber" : UInt, internal
   "DB_Machine_Sts_iStateID" : Int = PLC DB_Machine.Sts.iStateID AT %DB12.DBW4, 1 s
   "DB_Machine_Sts_iCurrentLayer" : Int = PLC DB_Machine.Sts.iCurrentLayer AT %DB12.DBW6, 1 s
   "DB_Machine_Sts_iTargetLayers" : Int = PLC DB_Machine.Sts.iTargetLayers AT %DB12.DBW8, 1 s
   "DB_Machine_Sts_xRunning" : Bool = PLC DB_Machine.Sts.xRunning AT %DB12.DBX2.2, 1 s
   "DB_Machine_Sts_xPaused" : Bool = PLC DB_Machine.Sts.xPaused AT %DB12.DBX2.3, 1 s
   "DB_Machine_Sts_xFaulted" : Bool = PLC DB_Machine.Sts.xFaulted AT %DB12.DBX2.4, 1 s
   "DB_Machine_Sts_xModeManual" : Bool = PLC DB_Machine.Sts.xModeManual AT %DB12.DBX2.1, 1 s
   "Cmd_Push_Manual" : Bool = PLC Cmd_Push_Manual AT %M0.7, 1 s
   "Cmd_Clamp_Manual" : Bool = PLC Cmd_Clamp_Manual AT %M3.1, 1 s
   "Cmd_Plate_Manual" : Bool = PLC Cmd_Plate_Manual AT %M3.3, 1 s
   "Cmd_ExitConv_Manual" : Bool = PLC Cmd_ExitConv_Manual AT %M4.1, 1 s
   "Cmd_BoxFeed_Manual" : Bool = PLC Cmd_BoxFeed_Manual AT %M3.7, 1 s
   "Cmd_PalletFeed_Auto" : Bool = PLC Cmd_PalletFeed_Auto AT %M3.5, 1 s
   "Cmd_PalletFeed_Manual" : Bool = PLC Cmd_PalletFeed_Manual AT %M4.0, 1 s
   "Cmd_ElevUp_Manual" : Bool = PLC Cmd_ElevUp_Manual AT %M4.3, 1 s
   "Cmd_ElevDown_Manual" : Bool = PLC Cmd_ElevDown_Manual AT %M4.5, 1 s
   "Cmd_Turn_Manual" : Bool = PLC Cmd_Turn_Manual AT %M4.7, 1 s
   "DB_Machine_Sts_iTotalBoxes" : DInt = PLC DB_Machine.Sts.iTotalBoxes AT %DB12.DBD10, 1 s
   "DB_Machine_Sts_iTotalPallets" : DInt = PLC DB_Machine.Sts.iTotalPallets AT %DB12.DBD14, 1 s
   "DB_Machine_Cmd_xHmiResetCounters" : Bool = PLC DB_Machine.Cmd.xHmiResetCounters AT %DB12.DBX0.6, 1 s
   "DB_Machine_Sts_wAlarmWord" : Word = PLC DB_Machine.Sts.wAlarmWord AT %DB12.DBW18, 500 ms
   "I_Reset" : Bool = PLC I_Reset AT %I1.5, 1 s
   "DB_Machine_Cmd_xHmiAckFault" : Bool = PLC DB_Machine.Cmd.xHmiAckFault AT %DB12.DBX0.7, 1 s
   "Cmd_BoxFeed_Auto" : Bool = PLC Cmd_BoxFeed_Auto AT %M3.4, 1 s

discrete alarms
   1: 'Fault ID 1: E-Stop Pressed', class Errors, trigger "DB_Machine_Sts_wAlarmWord" bit 1
   2: 'Fault ID 2: Pusher Timeout', class Errors, trigger "DB_Machine_Sts_wAlarmWord" bit 2
   3: 'Fault ID 3: Plate Timeout', class Errors, trigger "DB_Machine_Sts_wAlarmWord" bit 3
   4: 'Fault ID 4: Eject Timeout', class Errors, trigger "DB_Machine_Sts_wAlarmWord" bit 4

text list "Machine_States": 1 'OFF / IDLE'; 2 'AUTO RUNNING'; 3 'AUTO PAUSED'; 4 'MANUAL MODE'; 5 'FAULT ACTIVE'

screen "Root screen" 800x480, template "Template_1"
   on GenerateScreen: SetTag("Tag_ScreenNumber", 1)
   SymbolicIOField "Symbolic I/O field_2" at 549,211 size 178x32; TextOff '0'; TextOn '1'; TextList "Machine_States"
      ProcessValue <- "DB_Machine_Sts_iStateID"
   TextField "Text field_1" at 539,306 size 123x23; Text 'Current Layer:'
   TextField "Text field_2" at 538,341 size 124x23; Text 'Target Layers:'
   IOField "I/O field_1" at 676,304 size 46x32; FormatPattern 9
      ProcessValue <- "DB_Machine_Sts_iCurrentLayer"
   IOField "I/O field_2" at 676,340 size 46x32; FormatPattern 9
      ProcessValue <- "DB_Machine_Sts_iTargetLayers"
   Circle "Circle_1" at 627,47 size 48x48
      Appearance <- "DB_Machine_Sts_xPaused"
   Circle "Circle_2" at 537,47 size 48x48
      Appearance <- "DB_Machine_Sts_xRunning"
   Circle "Circle_3" at 710,47 size 48x48
      Appearance <- "DB_Machine_Sts_xFaulted"
   TextField "Text field_3" at 517,101 size 84x23; Text 'RUNNING'
   TextField "Text field_4" at 619,101 size 72x23; Text 'PAUSED'
   TextField "Text field_5" at 710,101 size 58x23; Text 'FAULT'
   Button "Button_1" at 541,146 size 192x53; TextOff 'MANUAL OVERRIDES'; Authorization "User administration"
      on Press: ActivateScreen("Screen_Manual", 0)
      Visibility <- "DB_Machine_Sts_xModeManual"
   TextField "Text field_6" at 553,400 size 108x23; Text 'Total Boxes:'
   TextField "Text field_7" at 552,435 size 115x23; Text 'Total Pallets:'
   IOField "I/O field_3" at 678,397 size 46x32; FormatPattern 9999999
      ProcessValue <- "DB_Machine_Sts_iTotalBoxes"
   IOField "I/O field_4" at 677,434 size 46x32; FormatPattern 9999999999
      ProcessValue <- "DB_Machine_Sts_iTotalPallets"
   AlarmView "Alarm view_1" at 25,89 size 466x377
   TextField "Text field_8" at 53,61 size 97x23; Text 'Alarm view'
   Button "Button_2" at 282,55 size 197x32; TextOff 'ACKNOWLEDGE FAULT'
      on Press: SetBit("DB_Machine_Cmd_xHmiAckFault")
      on Release: ResetBit("DB_Machine_Cmd_xHmiAckFault")
      Visibility <- "DB_Machine_Sts_xFaulted"

Template "Template_1" 800x480
   SymbolicIOField "Symbolic_IO_Field_Screen" at 93,9 size 600x33; TextOff '0'; TextOn '1'; TextList "TextList_ScreenNames"
      ProcessValue <- "Tag_ScreenNumber"
      on Change: ActivateScreenByNumber("Tag_ScreenNumber", 0)
   DateTimeField "HmiScreenItemData" at 695,25 size 105x25
   DateTimeField "HmiScreenItemData_1" at 695,0 size 105x25
   GraphicView "Logo" at 0,0 size 91x51; Picture "Logo of HMI_1"

screen "Screen_Manual" 800x480
   Button "Button_1" at 669,435 size 129x43; TextOff 'BACK TO MAIN'
      on Press: ActivateScreen("Root screen", 0)
   Button "Button_2" at 188,97 size 96x32; TextOff 'Pusher'
      on Press: SetBit("Cmd_Push_Manual")
      on Release: ResetBit("Cmd_Push_Manual")
   Button "Button_3" at 188,137 size 96x32; TextOff 'Plate'
      on Release: ResetBit("Cmd_Plate_Manual")
      on Press: SetBit("Cmd_Plate_Manual")
   Button "Button_4" at 188,182 size 96x32; TextOff 'Clamp'
      on Release: ResetBit("Cmd_Clamp_Manual")
      on Press: SetBit("Cmd_Clamp_Manual")
   Button "Button_5" at 469,137 size 120x34; TextOff 'Exit Motor'
      on Release: ResetBit("Cmd_ExitConv_Manual")
      on Press: SetBit("Cmd_ExitConv_Manual")
   Button "Button_6" at 469,177 size 120x37; TextOff 'Pallets Motor'
      on Release: ResetBit("Cmd_PalletFeed_Manual")
      on Press: SetBit("Cmd_PalletFeed_Manual")
   Button "Button_7" at 469,97 size 120x35; TextOff 'Boxs Motor'
      on Release: ResetBit("Cmd_BoxFeed_Manual")
      on Press: SetBit("Cmd_BoxFeed_Manual")
   Button "Button_8" at 469,225 size 120x35; TextOff 'Elevator UP'
      on Press: SetBit("Cmd_ElevUp_Manual")
      on Release: ResetBit("Cmd_ElevUp_Manual")
   Button "Button_9" at 469,273 size 120x34; TextOff 'Elevator Down'
      on Release: ResetBit("Cmd_ElevDown_Manual")
      on Press: SetBit("Cmd_ElevDown_Manual")
   Button "Button_10" at 187,223 size 97x32; TextOff 'Turn'
      on Release: ResetBit("Cmd_Turn_Manual")
      on Press: SetBit("Cmd_Turn_Manual")
   TextField "Text field_1" at 211,2 size 442x28; Text 'Manual mode for Testing and Maintenance'
   Circle "Circle_1" at 306,95 size 38x38
      Appearance <- "Cmd_Push_Manual"
   Circle "Circle_2" at 306,135 size 38x38
      Appearance <- "Cmd_Plate_Manual"
   Circle "Circle_3" at 306,177 size 38x38
      Appearance <- "Cmd_Clamp_Manual"
   Circle "Circle_4" at 306,217 size 38x38
      Appearance <- "Cmd_Turn_Manual"
   TextField "Text field_2" at 181,63 size 164x23; Text 'Pneumatic Controls'
   TextField "Text field_3" at 487,63 size 134x23; Text 'Motors Controls'
   Circle "Circle_5" at 599,98 size 38x38
      Appearance <- "Cmd_BoxFeed_Manual"
   Circle "Circle_6" at 599,141 size 38x38
      Appearance <- "Cmd_ExitConv_Manual"
   Circle "Circle_7" at 599,183 size 38x38
      Appearance <- "Cmd_PalletFeed_Manual"
   Circle "Circle_8" at 599,225 size 38x38
      Appearance <- "Cmd_ElevUp_Manual"
   Circle "Circle_9" at 599,270 size 38x38
      Appearance <- "Cmd_ElevDown_Manual"
   Button "Button_11" at 250,332 size 284x58; TextOff 'RESET COUNTERS & SEQUENCE'
      on Press: SetBit("DB_Machine_Cmd_xHmiResetCounters")
      on Release: ResetBit("DB_Machine_Cmd_xHmiResetCounters")

screen "Screen_1" 800x480
   GraphicView "Graphic view_1" at 63,84 size 225x64; Picture "Graphic_12"
*)